{attribute 'linkalways'}
{attribute 'hide_all_locals'}
FUNCTION_BLOCK ValueSintRead EXTENDS ValueBase IMPLEMENTS ValueRead
VAR
	thisValue : SINT;
END_VAR

{attribute 'call_after_global_init_slot' := '1'}
{attribute 'call_after_online_change_slot' := '1'}
METHOD PROTECTED GetThisAnyType
VAR_INPUT
END_VAR
thisAnyType := ToAnyType(thisValue);
END_METHOD

METHOD GetAsType : BOOL
VAR_INPUT
	destination : __SYSTEM.AnyType;
END_VAR
GetAsType := ConvertAnyType(thisAnyType, destination);
END_METHOD

METHOD GetAsString : T_MaxString
VAR_INPUT
END_VAR
GetAsString := TO_STRING(thisValue);
END_METHOD

METHOD Get : BOOL
VAR_INPUT
	destination : ANY;
END_VAR
Get := ConvertAnyType(thisAnyType, destination);
END_METHOD

METHOD FB_init : BOOL
VAR_INPUT
	bInitRetains : BOOL; // if TRUE, the retain variables are initialized (warm start / cold start)
	bInCopyCode : BOOL;  // if TRUE, the instance afterwards gets moved into the copy code (online change)
END_VAR
_ValueType := __SYSTEM.TYPE_CLASS.TYPE_SINT;
END_METHOD

{attribute 'monitoring' := 'call'}
PROPERTY Value : SINT
GET
Value := thisValue;
END_GET
END_PROPERTY

END_FUNCTION_BLOCK

(* stored: Version 1.1.0.1
   POU ValueSintRead: Id {40309194-f56f-4203-a8b1-122593d2f09a}, SpecialFunc None
   Method GetThisAnyType: Id {96fd8848-178b-4e30-9f3b-c17c34a0ff23}
   Method GetAsType: Id {468a0573-b53e-4bc6-b3ee-58d5f8d6e697}
   Method GetAsString: Id {5b05074a-0262-4f60-b9e5-4fca655158f3}
   Method Get: Id {e64175e4-41ee-48e9-b04f-febec47034f9}
   Method FB_init: Id {30a6c7bf-ec66-4290-af6f-64cfcff8c327}
   Property Value: Id {a0977e00-7afa-4bbb-a823-9deffd5005d3}
   Get Get: Id {95714049-8bed-462e-bd01-b29e73394f11} *)
